FUNCTION_BLOCK BUTTONAdp (* Composite Function Block Type *)
  (* Standard: 61499-2 *)
  (* Version 0.0, 7/20/2013, vvya002, nxtControl GmbH, template *)
  PACKAGE Main;
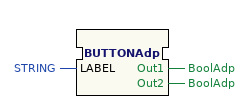
  VAR_INPUT
    LABEL : STRING;
  END_VAR
  PLUGS
    Out1 : BoolAdp;
    Out2 : BoolAdp;
  END_PLUGS
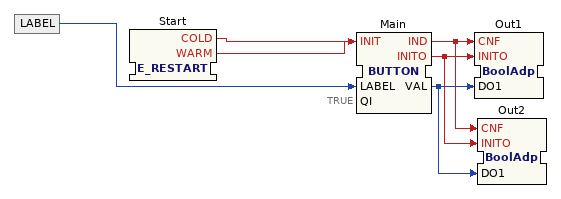
  FBS
    Main : BUTTON(QI := TRUE);
    Start : E_RESTART;
  END_FBS
  EVENT_CONNECTIONS
    Start.COLD TO Main.INIT;
    Start.WARM TO Main.INIT;
    Main.IND TO Out1.CNF;
    Main.IND TO Out2.CNF;
    Main.INITO TO Out1.INITO;
    Main.INITO TO Out2.INITO;
  END_CONNECTIONS
  DATA_CONNECTIONS
    LABEL TO Main.LABEL;
    Main.VAL TO Out1.DO1;
    Main.VAL TO Out2.DO1;
  END_CONNECTIONS
END_FUNCTION_BLOCK
